// TIA Portal V21 export
VAR_GLOBAL   // PLC tag table "Merker"
   Clock_1Hz AT %M1.5 : Bool;
   FirstScan AT %M0.0 : Bool;
END_VAR
